// TIA Portal project "TRAFFIC" (V16)

(* hardware
DEVICE "S7-1200 station_1"  S7-1200 Station
   slot 0: "Rack_0"  S7-1200 Rack  Rack  V1.0
   slot 1: "PLC_1"  CPU 1212C AC/DC/Rly  6ES7 212-1BE40-0XB0  V4.4
*)

// ===== PLC "PLC_1"  CPU 1212C AC/DC/Rly =====

VAR_GLOBAL   // PLC tag table "Default tag table"
   "START" AT %I0.0 : Bool;
   "STOP" AT %I0.1 : Bool;
   "MOTOR1" AT %Q0.0 : Bool;
   "MOTOR2" AT %Q0.1 : Bool;
   "MOTOR3" AT %Q0.2 : Bool;
   "MARKER X" AT %M0.0 : Bool;
   "MARKER Y" AT %M0.1 : Bool;
   "MARKER Z" AT %M0.2 : Bool;
   "Tag_1" AT %M0.3 : Bool;
END_VAR

// folder: System blocks/Program resources

DATA_BLOCK "TIMER1"   // DB1
{ S7_Optimized_Access := 'TRUE' }
AUTHOR : Simatic
FAMILY : IEC
NAME : IEC_TMR
VERSION : 1.0
// stored: InstanceOfName IEC_TIMER
"IEC_TIMER"
BEGIN
END_DATA_BLOCK

// folder: (top level)

ORGANIZATION_BLOCK "Main"   // OB1, LAD, ProgramCycle
TITLE = "Main Program Sweep (Cycle)"
{ S7_Optimized_Access := 'TRUE' }
VERSION : 0.1
   VAR_INPUT
      Initial_Call : Bool;   // Initial call of this OB
      Remanence : Bool;   // =True, if remanent data are available
   END_VAR
BEGIN

REGION Network 1
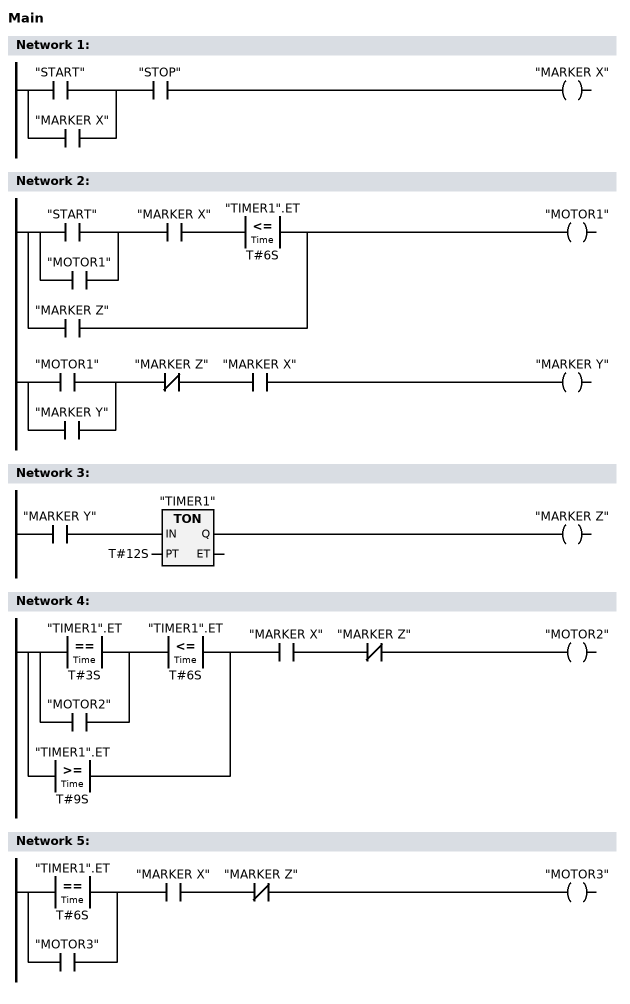
   RUNG wire#powerrail
      Contact( "START" )
      wire#w1
      Contact( "STOP" )
      Coil( "MARKER X" )
   END_RUNG
   RUNG wire#powerrail
      Contact( "MARKER X" )
   END_RUNG wire#w1
   // the same network as SCL:
   "MARKER X" := ("START" OR "MARKER X") AND "STOP";
END_REGION

REGION Network 2
   RUNG wire#powerrail
      Contact( "START" )
      wire#w1
      Contact( "MARKER X" )
      { S7_Templates := "SrcType := Time" } LE_Contact(in1 := "TIMER1".ET, in2 := T#6S)
      wire#w2
      Coil( "MOTOR1" )
   END_RUNG
   RUNG wire#powerrail
      Contact( "MOTOR1" )
   END_RUNG wire#w1
   RUNG wire#powerrail
      Contact( "MARKER Z" )
   END_RUNG wire#w2
   RUNG wire#powerrail
      Contact( "MOTOR1" )
      wire#w3
      I_Contact( "MARKER Z" )
      Contact( "MARKER X" )
      Coil( "MARKER Y" )
   END_RUNG
   RUNG wire#powerrail
      Contact( "MARKER Y" )
   END_RUNG wire#w3
   // the same network as SCL:
   "MOTOR1" := (("START" OR "MOTOR1") AND "MARKER X" AND ("TIMER1".ET <= T#6S)) OR "MARKER Z";
   "MARKER Y" := ("MOTOR1" OR "MARKER Y") AND NOT "MARKER Z" AND "MARKER X";
END_REGION

REGION Network 3
   "TIMER1".TON(IN := "MARKER Y", PT := T#12S);
   "MARKER Z" := "TIMER1".Q;
END_REGION

REGION Network 4
   RUNG wire#powerrail
      { S7_Templates := "SrcType := Time" } EQ_Contact(in1 := "TIMER1".ET, in2 := T#3S)
      wire#w1
      { S7_Templates := "SrcType := Time" } LE_Contact(in1 := "TIMER1".ET, in2 := T#6S)
      wire#w2
      Contact( "MARKER X" )
      I_Contact( "MARKER Z" )
      Coil( "MOTOR2" )
   END_RUNG
   RUNG wire#powerrail
      Contact( "MOTOR2" )
   END_RUNG wire#w1
   RUNG wire#powerrail
      { S7_Templates := "SrcType := Time" } GE_Contact(in1 := "TIMER1".ET, in2 := T#9S)
   END_RUNG wire#w2
   // the same network as SCL:
   "MOTOR2" := (((("TIMER1".ET = T#3S) OR "MOTOR2") AND ("TIMER1".ET <= T#6S)) OR ("TIMER1".ET >= T#9S)) AND "MARKER X" AND NOT "MARKER Z";
END_REGION

REGION Network 5
   RUNG wire#powerrail
      { S7_Templates := "SrcType := Time" } EQ_Contact(in1 := "TIMER1".ET, in2 := T#6S)
      wire#w1
      Contact( "MARKER X" )
      I_Contact( "MARKER Z" )
      Coil( "MOTOR3" )
   END_RUNG
   RUNG wire#powerrail
      Contact( "MOTOR3" )
   END_RUNG wire#w1
   // the same network as SCL:
   "MOTOR3" := (("TIMER1".ET = T#6S) OR "MOTOR3") AND "MARKER X" AND NOT "MARKER Z";
END_REGION
END_ORGANIZATION_BLOCK